TYPE ST_GC_DVID :
STRUCT
END_STRUCT
END_TYPE

(* stored: Version 1.1.0.1, ProductVersion 3.1.4026.18
   DUT ST_GC_DVID: Id {0471da07-3ebf-4173-9031-44630d98b9fd} *)
